{attribute addProperty BoxType "KL1004-0050"}
{attribute addProperty Id "Channel_1Channel_70B606D100Channel_2Channel_70B606D100Channel_3Channel_70B606D100Channel_4Channel_70B606D100Channel_5Channel_70B606D100Channel_6Channel_70B606D100Channel_7Channel_70B606D100Channel_8Channel_70B606D100Channel_9Channel_70B606D100Channel_10Channel_70B606D100Channel_11Channel_70B606D100Channel_12Channel_70B606D100Channel_13Channel_70B606D100Channel_14Channel_70B606D100Channel_15Channel_70B606D100Channel_16Channel_70B606D100Channel_17Channel_70B606D100Channel_18Channel_70B606D100Channel_19Channel_70B606D100Channel_20Channel_70B606D100Channel_21Channel_70B606D100Channel_22Channel_70B606D100Channel_23Channel_70B606D100Channel_24Channel_70B606D100Channel_25Channel_70B606D100Channel_26Channel_70B606D100Channel_27Channel_70B606D100Channel_28Channel_70B606D100Channel_29Channel_70B606D100Channel_30Channel_70B606D100Channel_31Channel_70B606D100Channel_32Channel_70B606D100"}
{attribute addProperty CRC "569132605"}
{attribute addProperty SizeInBites "0"}
{attribute addProperty SizeInBytes "0"}
TYPE KL_21EC463D :
STRUCT
	{attribute addProperty Name "Channel_1"}
	Channel_1 : Channel_70B606D1;
	{attribute addProperty Name "Channel_2"}
	Channel_2 : Channel_70B606D1;
	{attribute addProperty Name "Channel_3"}
	Channel_3 : Channel_70B606D1;
	{attribute addProperty Name "Channel_4"}
	Channel_4 : Channel_70B606D1;
	{attribute addProperty Name "Channel_5"}
	Channel_5 : Channel_70B606D1;
	{attribute addProperty Name "Channel_6"}
	Channel_6 : Channel_70B606D1;
	{attribute addProperty Name "Channel_7"}
	Channel_7 : Channel_70B606D1;
	{attribute addProperty Name "Channel_8"}
	Channel_8 : Channel_70B606D1;
	{attribute addProperty Name "Channel_9"}
	Channel_9 : Channel_70B606D1;
	{attribute addProperty Name "Channel_10"}
	Channel_10 : Channel_70B606D1;
	{attribute addProperty Name "Channel_11"}
	Channel_11 : Channel_70B606D1;
	{attribute addProperty Name "Channel_12"}
	Channel_12 : Channel_70B606D1;
	{attribute addProperty Name "Channel_13"}
	Channel_13 : Channel_70B606D1;
	{attribute addProperty Name "Channel_14"}
	Channel_14 : Channel_70B606D1;
	{attribute addProperty Name "Channel_15"}
	Channel_15 : Channel_70B606D1;
	{attribute addProperty Name "Channel_16"}
	Channel_16 : Channel_70B606D1;
	{attribute addProperty Name "Channel_17"}
	Channel_17 : Channel_70B606D1;
	{attribute addProperty Name "Channel_18"}
	Channel_18 : Channel_70B606D1;
	{attribute addProperty Name "Channel_19"}
	Channel_19 : Channel_70B606D1;
	{attribute addProperty Name "Channel_20"}
	Channel_20 : Channel_70B606D1;
	{attribute addProperty Name "Channel_21"}
	Channel_21 : Channel_70B606D1;
	{attribute addProperty Name "Channel_22"}
	Channel_22 : Channel_70B606D1;
	{attribute addProperty Name "Channel_23"}
	Channel_23 : Channel_70B606D1;
	{attribute addProperty Name "Channel_24"}
	Channel_24 : Channel_70B606D1;
	{attribute addProperty Name "Channel_25"}
	Channel_25 : Channel_70B606D1;
	{attribute addProperty Name "Channel_26"}
	Channel_26 : Channel_70B606D1;
	{attribute addProperty Name "Channel_27"}
	Channel_27 : Channel_70B606D1;
	{attribute addProperty Name "Channel_28"}
	Channel_28 : Channel_70B606D1;
	{attribute addProperty Name "Channel_29"}
	Channel_29 : Channel_70B606D1;
	{attribute addProperty Name "Channel_30"}
	Channel_30 : Channel_70B606D1;
	{attribute addProperty Name "Channel_31"}
	Channel_31 : Channel_70B606D1;
	{attribute addProperty Name "Channel_32"}
	Channel_32 : Channel_70B606D1;
END_STRUCT
END_TYPE

(* stored: Version 1.2.0.0, ProductVersion 3.1.4024.9
   DUT KL_21EC463D: Id {396448d0-811a-4222-97a9-99bdf8eca6bd} *)
